Omron Sysmac Studio project CSV Test (Sysmac Studio 1.40.0.64008, StandardProject)

# Controller new_Controller_0: NX102-1020 version 1.34
Task PrimaryTask (priority 4, period or condition 2000): Program0

TYPE RobPosTM12 : STRUCT
    RobPosX : STRING[255];
    RobPosY : STRING[255];
    RobPosZ : STRING[255];
    RobPosRx : STRING[255];
    RobPosRy : STRING[255];
    RobPosRz : STRING[255];
END_STRUCT END_TYPE

VAR_GLOBAL
    RobPos : ARRAY[0..5] OF REAL;
    RobPosTM : array[0..7] of RobPosTM12;
END_VAR

PROGRAM Program0
VAR
    TrigRoboProgramRead : BOOL;
    ProgramToOpen : STRING[255];
    OpenRoboProgram : FileOpen;
    ReadRoboProgram : FileGets;
    Fid : DWORD;
    Index : DINT;
    InDat : ARRAY[0..254] OF INT;
    CloseRoboProgram : FileClose;
    ReadComplete : BOOL;
    OpenFileError : BOOL;
    CloseFileError : BOOL;
    ReadFileError : BOOL;
    AIndex : DINT;
    test : BOOL;
END_VAR
VAR_EXTERNAL
    RobPosTM : array[0..7] of RobPosTM12;
END_VAR
VAR
    _p1 : BOOL;
    _p2 : BOOL;
    _e3 : R_TRIG;
END_VAR

(* Section Section0: ladder, written here as Structured Text *)

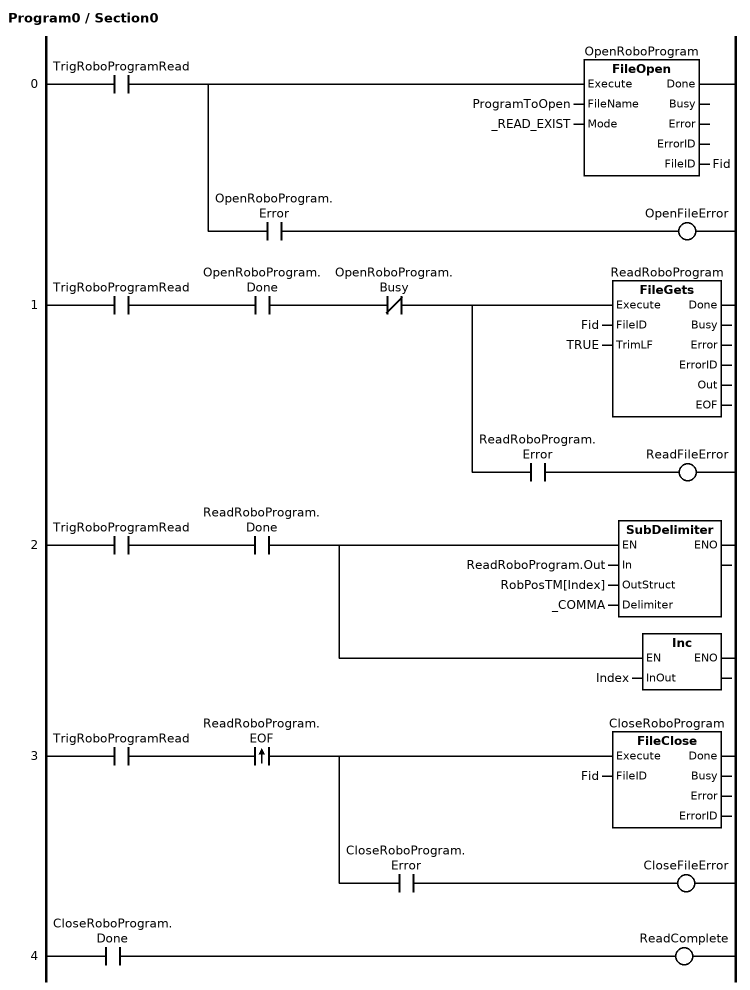
(* Rung 0 *)
OpenRoboProgram(Execute := TrigRoboProgramRead, FileName := ProgramToOpen, Mode := _READ_EXIST, FileID => Fid);
OpenFileError := TrigRoboProgramRead AND OpenRoboProgram.Error;
(* Rung 1 *)
_p1 := TrigRoboProgramRead AND OpenRoboProgram.Done AND NOT OpenRoboProgram.Busy;
ReadRoboProgram(Execute := _p1, FileID := Fid, TrimLF := TRUE);
ReadFileError := _p1 AND ReadRoboProgram.Error;
(* Rung 2 *)
_p2 := TrigRoboProgramRead AND ReadRoboProgram.Done;
IF _p2 THEN
    SubDelimiter(In := ReadRoboProgram.Out, OutStruct := RobPosTM[Index], Delimiter := _COMMA);
    Inc(InOut := Index);
END_IF;
(* Rung 3 *)
_e3(CLK := ReadRoboProgram.EOF);
CloseRoboProgram(Execute := TrigRoboProgramRead AND _e3.Q, FileID := Fid);
CloseFileError := TrigRoboProgramRead AND _e3.Q AND CloseRoboProgram.Error;
(* Rung 4 *)
ReadComplete := CloseRoboProgram.Done;
END_PROGRAM